{attribute addProperty BoxType "BK1250-0000-0018"}
{attribute addProperty Id "Term_389_KL1002KL1002_D229A9CA00"}
{attribute addProperty CRC "2519066313"}
{attribute addProperty SizeInBites "0"}
{attribute addProperty SizeInBytes "0"}
TYPE A_0017_BK1250_0000_0018_9625E6C9 EXTENDS BK1250_4487A81F :
STRUCT
	{attribute addProperty Name "Term_389_KL1002"}
	Term_389_KL1002 : KL1002_D229A9CA;
END_STRUCT
END_TYPE

(* stored: Version 1.2.0.0, ProductVersion 3.1.4024.9
   DUT A_0017_BK1250_0000_0018_9625E6C9: Id {dbe9a101-9ed4-4227-a9f8-b01aab36ebb9} *)
